Staubli VAL3: onStart.pgx

program onStart(bool& x_bResult[])
  local num i
  local num l_nIndex
  local num l_nSize
  local string l_sMessage[2]
  local bool l_bOk
begin
  cls()
  userPage()
  call use:nullKey(nKey)
  call buildList()
  call refreshStatic()
  x_bResult=true
end
